// TIA Portal V20 export
DATA_BLOCK "ControlNodes"   // DB114
// stored: MemoryReserve 100, Namespace Unit1.Em6
   VAR
      em { ExternalWritable := 'False'} : "LAF_typeEmControlNode";
      cm { ExternalWritable := 'False'} : "Unit1.Em6.typeCmControlNode";
      citiMap : "LER_OEM_Data";
      visionUnit { ExternalWritable := 'False'} : "Unit1.Em6.typeSequenceControlNode";
      visionController { ExternalWritable := 'False'} : "Unit1.Em6.typeSequenceControlNode";
      qrRead { ExternalWritable := 'False'} : "Unit1.Em6.typeSequenceControlNode";
   END_VAR
   VAR RETAIN
      cmVisionUnitAxisZ { ExternalWritable := 'False'} : "LBC_typeAxis64PosControlNode";
      cmVisionPusherSupportUpDown { ExternalWritable := 'False'} : "LBC_typeTwoWayActuatorControlNode";
      cmVisionTriggerSensor { ExternalWritable := 'False'} : "LBC_typeDigitalSignalControlNode";
      cmVisionController { ExternalWritable := 'False'} : "LER_typeVisionControlNode";
      cmQrReader { ExternalWritable := 'False'} : "LER_typeSRX300ControlNode";
      cmQrReadHandy { ExternalWritable := 'False'} : "LER_typeDM8700ControlNode";
      cmVisionUnitAxisZ_TorqueCal { ExternalWritable := 'False'} : "LER_typeServoTorqueCalControlNode";
   END_VAR
BEGIN
   // cm.brakeTest.visionUnit.monitoring.error : Vision Axis Brake Test Error
   // cm.brakeTest.visionUnit.monitoring.busy : Vision Axis Brake Test In progress
END_DATA_BLOCK
